DATA_BLOCK "ext"
{ S7_Optimized_Access := 'FALSE' }
VERSION : 0.1
NON_RETAIN
   STRUCT
      block : Bool;
      trig : USInt;
      selector : Array[1..32] of Bool;
      status : Array[1..32] of USInt;
   END_STRUCT;


BEGIN
   block := true;
   selector[1] := true;
   selector[3] := true;
   selector[7] := true;
   selector[8] := true;
   selector[9] := true;
   selector[15] := true;
   selector[16] := true;
   selector[17] := true;
   selector[18] := true;
   selector[19] := true;
   selector[20] := true;
   selector[21] := true;
   selector[22] := true;

END_DATA_BLOCK

